// TIA Portal V17 export
// export: Created 2024-09-02T12:50:26.1758554Z, ExportSetting WithDefaults, DisplayName Totally Integrated Automation Portal, DisplayVersion V17, DisplayName TIA Portal Openness, DisplayVersion V17, DisplayName TIA Portal Version Control Interface, DisplayVersion V17, DisplayName STEP 7 Professional, DisplayVersion V17, DisplayName STEP 7 Safety, DisplayVersion V17, DisplayName WinCC Professional, DisplayVersion V17
TYPE "type_HMI_Layout"
// stored: IsFailsafeCompliant false
   STRUCT
      Estop : Array[0..7] of Bool;
      LightCourtain : Array[0..7] of Int;
      Door : Array[0..7] of Int;
      Signailing : Array[0..7] of Struct
         Green : Int;
         Yellow : Int;
         Red : Int;
         White : Int;
         Blue : Int;
      END_STRUCT;
      PalletStatus : Array[0..7] of Int;
      DeviceStatus : Array[0..7] of Int;
   END_STRUCT;
END_TYPE
